// TIA Portal V17 export
// export: Created 2025-03-05T07:59:49.5409179Z, ExportSetting WithDefaults, DisplayName Totally Integrated Automation Portal, DisplayVersion V17 Update 8, DisplayName TIA Portal Openness, DisplayVersion V17 Update 8, DisplayName TIA Portal Version Control Interface, DisplayVersion V17, DisplayName SINAMICS Startdrive Advanced, DisplayVersion V17 SP2, DisplayName SINAMICS Startdrive G110M, G120, G120C, G120D, G120P, G115D, DisplayVersion V17 SP2, DisplayName SINAMICS Startdrive G130, G150, S120, S150, SINAMICS MV, S210, DisplayVersion V17 SP2, DisplayName STEP 7 Professional, DisplayVersion V17 Update 8, DisplayName SINUMERIK ONE STEP 7 Toolbox, DisplayVersion V17 Update 12, DisplayName SINUMERIK 840D sl STEP 7 Toolbox, DisplayVersion V17 Update 12, DisplayName STEP 7 Safety, DisplayVersion V17 Update 6, DisplayName WinCC Advanced, DisplayVersion V17 Update 8
FUNCTION "FC368_NCK_M_CH8_UNIT_03" : Void   // FC368, LAD
TITLE = Channel 1 data
{ S7_Optimized_Access := 'FALSE' }
AUTHOR : ETXETAR
VERSION : 1.0
// stored: AutoNumber false, IsIECCheckEnabled false, SetENOAutomatically false, UDAEnableTagReadback false
   VAR_TEMP
      auxm3 : Bool;
      auxm5 : Bool;
   END_VAR
   VAR_TEMP   // added for the SCL form of the ladder/FBD networks
      _w1 : Bool;
      _w2 : Bool;
   END_VAR
BEGIN

REGION Network 1: CALL FB331 M CODE EXTENDED CH4 / M CODE EXTENDED CHANNEL 2
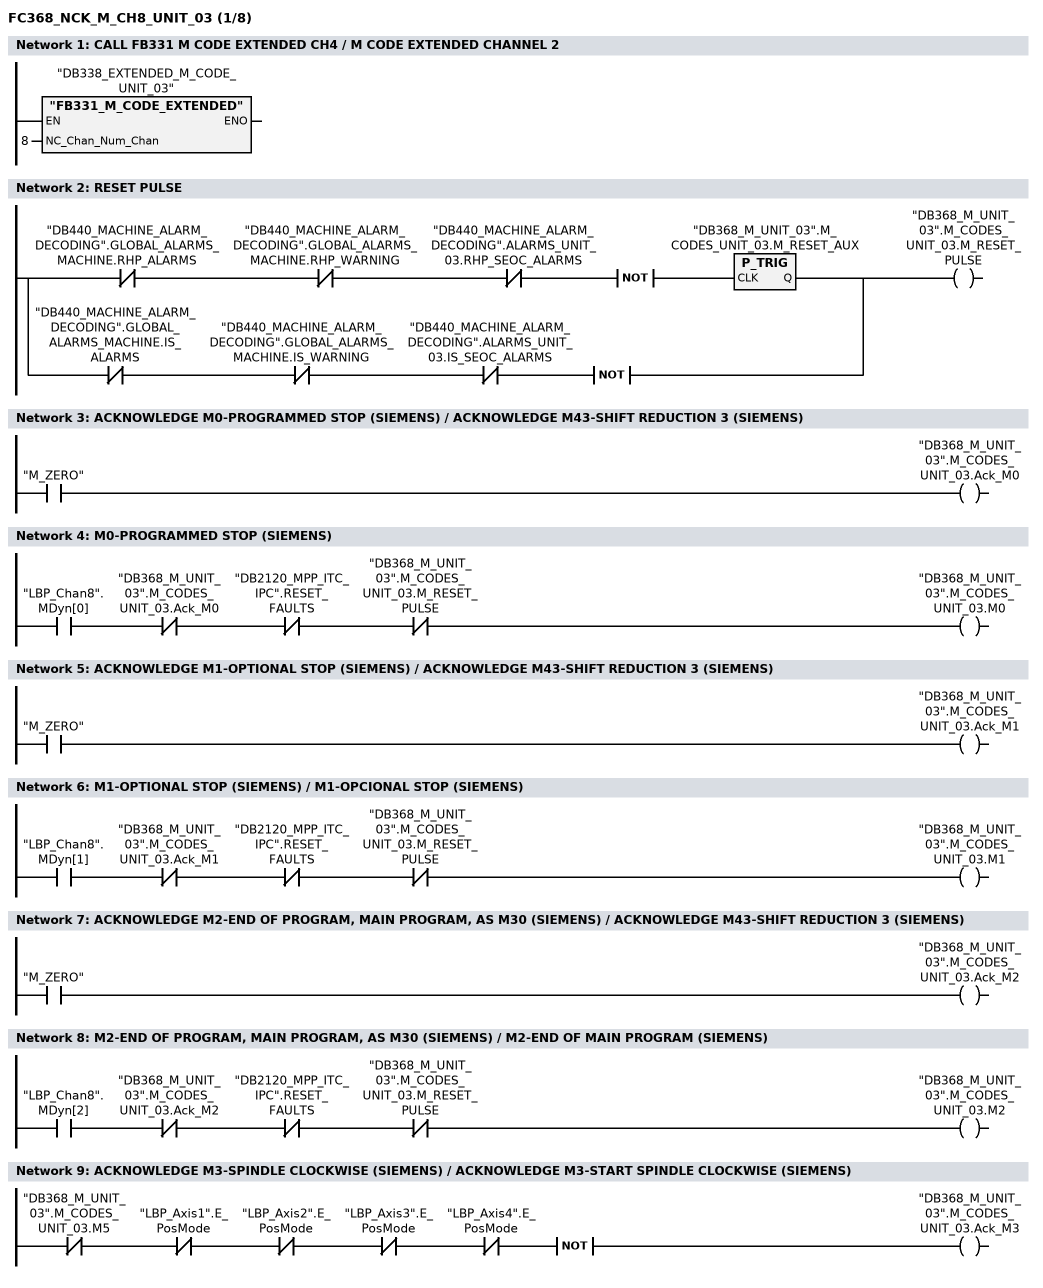
   RUNG wire#powerrail
      "DB338_EXTENDED_M_CODE_UNIT_03"(NC_Chan_Num_Chan := 8)
   END_RUNG
   // the same network as SCL:
   "DB338_EXTENDED_M_CODE_UNIT_03"(NC_Chan_Num_Chan := 8);   // "FB331_M_CODE_EXTENDED"
END_REGION

REGION Network 2: RESET PULSE
   RUNG wire#powerrail
      I_Contact( "DB440_MACHINE_ALARM_DECODING".GLOBAL_ALARMS_MACHINE.RHP_ALARMS )
      I_Contact( "DB440_MACHINE_ALARM_DECODING".GLOBAL_ALARMS_MACHINE.RHP_WARNING )
      I_Contact( "DB440_MACHINE_ALARM_DECODING".ALARMS_UNIT_03.RHP_SEOC_ALARMS )
      Not()
      P_Trig( "DB368_M_UNIT_03".M_CODES_UNIT_03.M_RESET_AUX )
      wire#w1
      Coil( "DB368_M_UNIT_03".M_CODES_UNIT_03.M_RESET_PULSE )
   END_RUNG
   RUNG wire#powerrail
      I_Contact( "DB440_MACHINE_ALARM_DECODING".GLOBAL_ALARMS_MACHINE.IS_ALARMS )
      I_Contact( "DB440_MACHINE_ALARM_DECODING".GLOBAL_ALARMS_MACHINE.IS_WARNING )
      I_Contact( "DB440_MACHINE_ALARM_DECODING".ALARMS_UNIT_03.IS_SEOC_ALARMS )
      Not()
   END_RUNG wire#w1
   // the same network as SCL:
   #_w1 := NOT (NOT "DB440_MACHINE_ALARM_DECODING".GLOBAL_ALARMS_MACHINE.RHP_ALARMS AND NOT "DB440_MACHINE_ALARM_DECODING".GLOBAL_ALARMS_MACHINE.RHP_WARNING AND NOT "DB440_MACHINE_ALARM_DECODING".ALARMS_UNIT_03.RHP_SEOC_ALARMS);
   #_w2 := #_w1 AND NOT "DB368_M_UNIT_03".M_CODES_UNIT_03.M_RESET_AUX;   // rising edge
   "DB368_M_UNIT_03".M_CODES_UNIT_03.M_RESET_AUX := #_w1;
   "DB368_M_UNIT_03".M_CODES_UNIT_03.M_RESET_PULSE := #_w2 OR NOT (NOT "DB440_MACHINE_ALARM_DECODING".GLOBAL_ALARMS_MACHINE.IS_ALARMS AND NOT "DB440_MACHINE_ALARM_DECODING".GLOBAL_ALARMS_MACHINE.IS_WARNING AND NOT "DB440_MACHINE_ALARM_DECODING".ALARMS_UNIT_03.IS_SEOC_ALARMS);
END_REGION

REGION Network 3: ACKNOWLEDGE M0-PROGRAMMED STOP (SIEMENS) / ACKNOWLEDGE M43-SHIFT REDUCTION 3 (SIEMENS)
   RUNG wire#powerrail
      Contact( "M_ZERO" )
      Coil( "DB368_M_UNIT_03".M_CODES_UNIT_03.Ack_M0 )
   END_RUNG
   // the same network as SCL:
   "DB368_M_UNIT_03".M_CODES_UNIT_03.Ack_M0 := "M_ZERO";
END_REGION

REGION Network 4: M0-PROGRAMMED STOP (SIEMENS)
   RUNG wire#powerrail
      Contact( "LBP_Chan8".MDyn[0] )
      I_Contact( "DB368_M_UNIT_03".M_CODES_UNIT_03.Ack_M0 )
      I_Contact( "DB2120_MPP_ITC_IPC".RESET_FAULTS )
      I_Contact( "DB368_M_UNIT_03".M_CODES_UNIT_03.M_RESET_PULSE )
      Coil( "DB368_M_UNIT_03".M_CODES_UNIT_03.M0 )
   END_RUNG
   // the same network as SCL:
   "DB368_M_UNIT_03".M_CODES_UNIT_03.M0 := "LBP_Chan8".MDyn[0] AND NOT "DB368_M_UNIT_03".M_CODES_UNIT_03.Ack_M0 AND NOT "DB2120_MPP_ITC_IPC".RESET_FAULTS AND NOT "DB368_M_UNIT_03".M_CODES_UNIT_03.M_RESET_PULSE;
END_REGION

REGION Network 5: ACKNOWLEDGE M1-OPTIONAL STOP (SIEMENS) / ACKNOWLEDGE M43-SHIFT REDUCTION 3 (SIEMENS)
   RUNG wire#powerrail
      Contact( "M_ZERO" )
      Coil( "DB368_M_UNIT_03".M_CODES_UNIT_03.Ack_M1 )
   END_RUNG
   // the same network as SCL:
   "DB368_M_UNIT_03".M_CODES_UNIT_03.Ack_M1 := "M_ZERO";
END_REGION

REGION Network 6: M1-OPTIONAL STOP (SIEMENS) / M1-OPCIONAL STOP (SIEMENS)
   RUNG wire#powerrail
      Contact( "LBP_Chan8".MDyn[1] )
      I_Contact( "DB368_M_UNIT_03".M_CODES_UNIT_03.Ack_M1 )
      I_Contact( "DB2120_MPP_ITC_IPC".RESET_FAULTS )
      I_Contact( "DB368_M_UNIT_03".M_CODES_UNIT_03.M_RESET_PULSE )
      Coil( "DB368_M_UNIT_03".M_CODES_UNIT_03.M1 )
   END_RUNG
   // the same network as SCL:
   "DB368_M_UNIT_03".M_CODES_UNIT_03.M1 := "LBP_Chan8".MDyn[1] AND NOT "DB368_M_UNIT_03".M_CODES_UNIT_03.Ack_M1 AND NOT "DB2120_MPP_ITC_IPC".RESET_FAULTS AND NOT "DB368_M_UNIT_03".M_CODES_UNIT_03.M_RESET_PULSE;
END_REGION

REGION Network 7: ACKNOWLEDGE M2-END OF PROGRAM, MAIN PROGRAM, AS M30 (SIEMENS) / ACKNOWLEDGE M43-SHIFT REDUCTION 3 (SIEMENS)
   RUNG wire#powerrail
      Contact( "M_ZERO" )
      Coil( "DB368_M_UNIT_03".M_CODES_UNIT_03.Ack_M2 )
   END_RUNG
   // the same network as SCL:
   "DB368_M_UNIT_03".M_CODES_UNIT_03.Ack_M2 := "M_ZERO";
END_REGION

REGION Network 8: M2-END OF PROGRAM, MAIN PROGRAM, AS M30 (SIEMENS) / M2-END OF MAIN PROGRAM (SIEMENS)
   RUNG wire#powerrail
      Contact( "LBP_Chan8".MDyn[2] )
      I_Contact( "DB368_M_UNIT_03".M_CODES_UNIT_03.Ack_M2 )
      I_Contact( "DB2120_MPP_ITC_IPC".RESET_FAULTS )
      I_Contact( "DB368_M_UNIT_03".M_CODES_UNIT_03.M_RESET_PULSE )
      Coil( "DB368_M_UNIT_03".M_CODES_UNIT_03.M2 )
   END_RUNG
   // the same network as SCL:
   "DB368_M_UNIT_03".M_CODES_UNIT_03.M2 := "LBP_Chan8".MDyn[2] AND NOT "DB368_M_UNIT_03".M_CODES_UNIT_03.Ack_M2 AND NOT "DB2120_MPP_ITC_IPC".RESET_FAULTS AND NOT "DB368_M_UNIT_03".M_CODES_UNIT_03.M_RESET_PULSE;
END_REGION

REGION Network 9: ACKNOWLEDGE M3-SPINDLE CLOCKWISE (SIEMENS) / ACKNOWLEDGE M3-START SPINDLE CLOCKWISE (SIEMENS)
   RUNG wire#powerrail
      I_Contact( "DB368_M_UNIT_03".M_CODES_UNIT_03.M5 )
      I_Contact( "LBP_Axis1".E_PosMode )
      I_Contact( "LBP_Axis2".E_PosMode )
      I_Contact( "LBP_Axis3".E_PosMode )
      I_Contact( "LBP_Axis4".E_PosMode )
      Not()
      Coil( "DB368_M_UNIT_03".M_CODES_UNIT_03.Ack_M3 )
   END_RUNG
   // the same network as SCL:
   "DB368_M_UNIT_03".M_CODES_UNIT_03.Ack_M3 := NOT (NOT "DB368_M_UNIT_03".M_CODES_UNIT_03.M5 AND NOT "LBP_Axis1".E_PosMode AND NOT "LBP_Axis2".E_PosMode AND NOT "LBP_Axis3".E_PosMode AND NOT "LBP_Axis4".E_PosMode);
END_REGION

REGION Network 10: M3-SPINDLE CLOCKWISE AUXILIARY (SIEMENS) / Extended address M function 1 (16 bit INT)
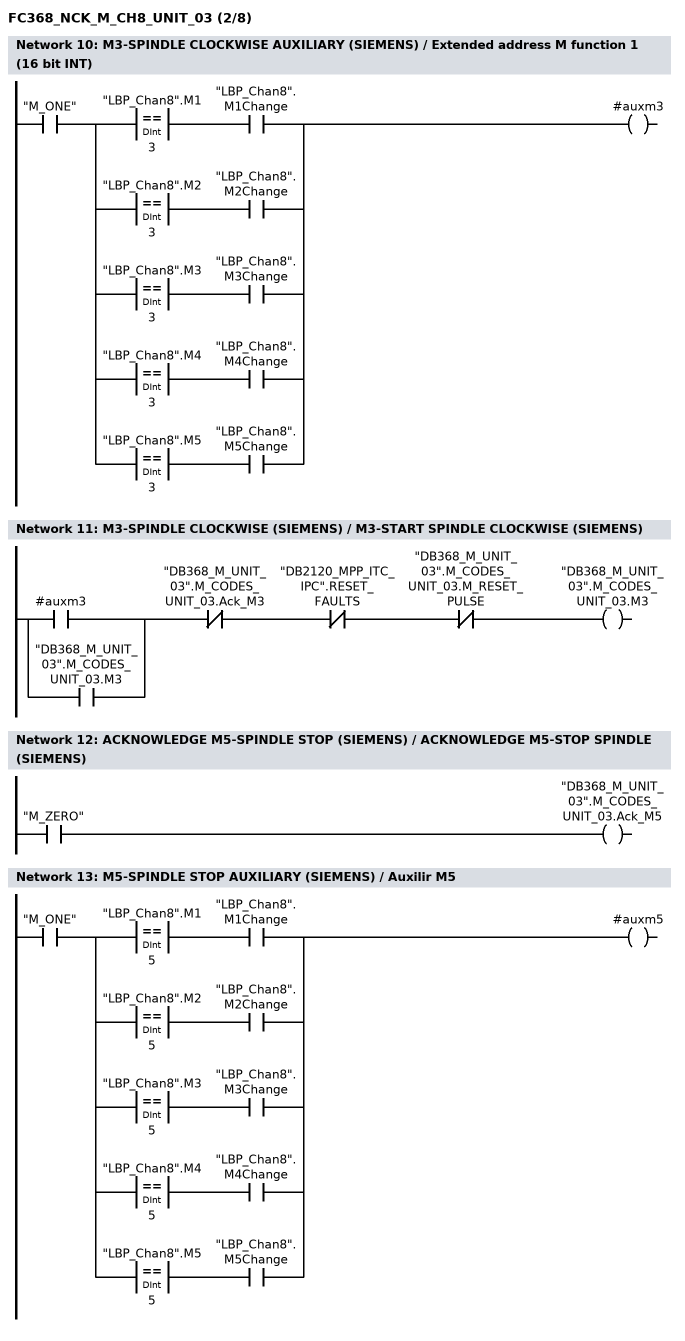
   RUNG wire#powerrail
      Contact( "M_ONE" )
      wire#w1
      { S7_Templates := "SrcType := DInt" } EQ_Contact(in1 := "LBP_Chan8".M1, in2 := 3)
      Contact( "LBP_Chan8".M1Change )
      wire#w2
      Coil( #auxm3 )
   END_RUNG
   RUNG wire#w1
      { S7_Templates := "SrcType := DInt" } EQ_Contact(in1 := "LBP_Chan8".M2, in2 := 3)
      Contact( "LBP_Chan8".M2Change )
   END_RUNG wire#w2
   RUNG wire#w1
      { S7_Templates := "SrcType := DInt" } EQ_Contact(in1 := "LBP_Chan8".M3, in2 := 3)
      Contact( "LBP_Chan8".M3Change )
   END_RUNG wire#w2
   RUNG wire#w1
      { S7_Templates := "SrcType := DInt" } EQ_Contact(in1 := "LBP_Chan8".M4, in2 := 3)
      Contact( "LBP_Chan8".M4Change )
   END_RUNG wire#w2
   RUNG wire#w1
      { S7_Templates := "SrcType := DInt" } EQ_Contact(in1 := "LBP_Chan8".M5, in2 := 3)
      Contact( "LBP_Chan8".M5Change )
   END_RUNG wire#w2
   // the same network as SCL:
   #auxm3 := "M_ONE" AND ((("LBP_Chan8".M1 = 3) AND "LBP_Chan8".M1Change) OR (("LBP_Chan8".M2 = 3) AND "LBP_Chan8".M2Change) OR (("LBP_Chan8".M3 = 3) AND "LBP_Chan8".M3Change) OR (("LBP_Chan8".M4 = 3) AND "LBP_Chan8".M4Change) OR (("LBP_Chan8".M5 = 3) AND "LBP_Chan8".M5Change));
END_REGION

REGION Network 11: M3-SPINDLE CLOCKWISE (SIEMENS) / M3-START SPINDLE CLOCKWISE (SIEMENS)
   RUNG wire#powerrail
      Contact( #auxm3 )
      wire#w1
      I_Contact( "DB368_M_UNIT_03".M_CODES_UNIT_03.Ack_M3 )
      I_Contact( "DB2120_MPP_ITC_IPC".RESET_FAULTS )
      I_Contact( "DB368_M_UNIT_03".M_CODES_UNIT_03.M_RESET_PULSE )
      Coil( "DB368_M_UNIT_03".M_CODES_UNIT_03.M3 )
   END_RUNG
   RUNG wire#powerrail
      Contact( "DB368_M_UNIT_03".M_CODES_UNIT_03.M3 )
   END_RUNG wire#w1
   // the same network as SCL:
   "DB368_M_UNIT_03".M_CODES_UNIT_03.M3 := (#auxm3 OR "DB368_M_UNIT_03".M_CODES_UNIT_03.M3) AND NOT "DB368_M_UNIT_03".M_CODES_UNIT_03.Ack_M3 AND NOT "DB2120_MPP_ITC_IPC".RESET_FAULTS AND NOT "DB368_M_UNIT_03".M_CODES_UNIT_03.M_RESET_PULSE;
END_REGION

REGION Network 12: ACKNOWLEDGE M5-SPINDLE STOP (SIEMENS) / ACKNOWLEDGE M5-STOP SPINDLE (SIEMENS)
   RUNG wire#powerrail
      Contact( "M_ZERO" )
      Coil( "DB368_M_UNIT_03".M_CODES_UNIT_03.Ack_M5 )
   END_RUNG
   // the same network as SCL:
   "DB368_M_UNIT_03".M_CODES_UNIT_03.Ack_M5 := "M_ZERO";
END_REGION

REGION Network 13: M5-SPINDLE STOP AUXILIARY (SIEMENS) / Auxilir M5
   RUNG wire#powerrail
      Contact( "M_ONE" )
      wire#w1
      { S7_Templates := "SrcType := DInt" } EQ_Contact(in1 := "LBP_Chan8".M1, in2 := 5)
      Contact( "LBP_Chan8".M1Change )
      wire#w2
      Coil( #auxm5 )
   END_RUNG
   RUNG wire#w1
      { S7_Templates := "SrcType := DInt" } EQ_Contact(in1 := "LBP_Chan8".M2, in2 := 5)
      Contact( "LBP_Chan8".M2Change )
   END_RUNG wire#w2
   RUNG wire#w1
      { S7_Templates := "SrcType := DInt" } EQ_Contact(in1 := "LBP_Chan8".M3, in2 := 5)
      Contact( "LBP_Chan8".M3Change )
   END_RUNG wire#w2
   RUNG wire#w1
      { S7_Templates := "SrcType := DInt" } EQ_Contact(in1 := "LBP_Chan8".M4, in2 := 5)
      Contact( "LBP_Chan8".M4Change )
   END_RUNG wire#w2
   RUNG wire#w1
      { S7_Templates := "SrcType := DInt" } EQ_Contact(in1 := "LBP_Chan8".M5, in2 := 5)
      Contact( "LBP_Chan8".M5Change )
   END_RUNG wire#w2
   // the same network as SCL:
   #auxm5 := "M_ONE" AND ((("LBP_Chan8".M1 = 5) AND "LBP_Chan8".M1Change) OR (("LBP_Chan8".M2 = 5) AND "LBP_Chan8".M2Change) OR (("LBP_Chan8".M3 = 5) AND "LBP_Chan8".M3Change) OR (("LBP_Chan8".M4 = 5) AND "LBP_Chan8".M4Change) OR (("LBP_Chan8".M5 = 5) AND "LBP_Chan8".M5Change));
END_REGION

REGION Network 14: M5-SPINDLE STOP (SIEMENS) / M5-STOP SPINDLE (SIEMENS)
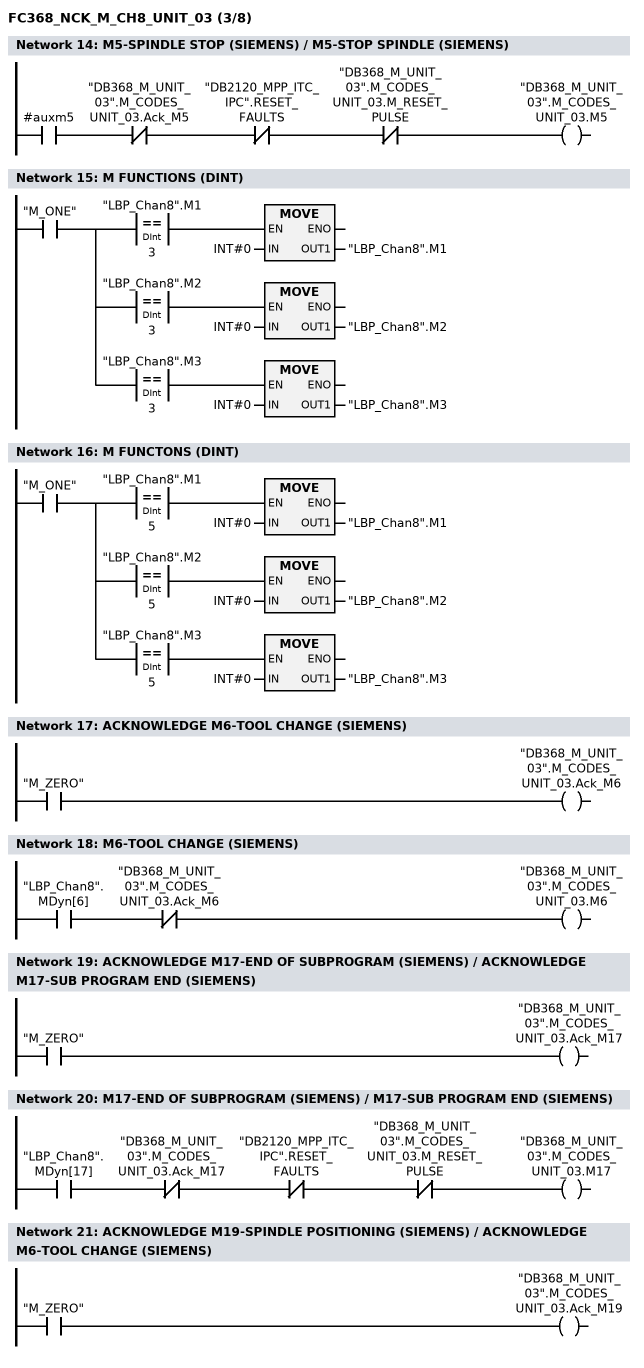
   RUNG wire#powerrail
      Contact( #auxm5 )
      I_Contact( "DB368_M_UNIT_03".M_CODES_UNIT_03.Ack_M5 )
      I_Contact( "DB2120_MPP_ITC_IPC".RESET_FAULTS )
      I_Contact( "DB368_M_UNIT_03".M_CODES_UNIT_03.M_RESET_PULSE )
      Coil( "DB368_M_UNIT_03".M_CODES_UNIT_03.M5 )
   END_RUNG
   // the same network as SCL:
   "DB368_M_UNIT_03".M_CODES_UNIT_03.M5 := #auxm5 AND NOT "DB368_M_UNIT_03".M_CODES_UNIT_03.Ack_M5 AND NOT "DB2120_MPP_ITC_IPC".RESET_FAULTS AND NOT "DB368_M_UNIT_03".M_CODES_UNIT_03.M_RESET_PULSE;
END_REGION

REGION Network 15: M FUNCTIONS (DINT)
   RUNG wire#powerrail
      Contact( "M_ONE" )
      wire#w1
      { S7_Templates := "SrcType := DInt" } EQ_Contact(in1 := "LBP_Chan8".M1, in2 := 3)
      { S7_GenerateENO := "TRUE" } Move(in := INT#0, out1 => "LBP_Chan8".M1)
   END_RUNG
   RUNG wire#w1
      { S7_Templates := "SrcType := DInt" } EQ_Contact(in1 := "LBP_Chan8".M2, in2 := 3)
      { S7_GenerateENO := "TRUE" } Move(in := INT#0, out1 => "LBP_Chan8".M2)
   END_RUNG
   RUNG wire#w1
      { S7_Templates := "SrcType := DInt" } EQ_Contact(in1 := "LBP_Chan8".M3, in2 := 3)
      { S7_GenerateENO := "TRUE" } Move(in := INT#0, out1 => "LBP_Chan8".M3)
   END_RUNG
   // the same network as SCL:
   IF "M_ONE" AND ("LBP_Chan8".M1 = 3) THEN "LBP_Chan8".M1 := INT#0; END_IF;
   IF "M_ONE" AND ("LBP_Chan8".M2 = 3) THEN "LBP_Chan8".M2 := INT#0; END_IF;
   IF "M_ONE" AND ("LBP_Chan8".M3 = 3) THEN "LBP_Chan8".M3 := INT#0; END_IF;
END_REGION

REGION Network 16: M FUNCTONS (DINT)
   RUNG wire#powerrail
      Contact( "M_ONE" )
      wire#w1
      { S7_Templates := "SrcType := DInt" } EQ_Contact(in1 := "LBP_Chan8".M1, in2 := 5)
      { S7_GenerateENO := "TRUE" } Move(in := INT#0, out1 => "LBP_Chan8".M1)
   END_RUNG
   RUNG wire#w1
      { S7_Templates := "SrcType := DInt" } EQ_Contact(in1 := "LBP_Chan8".M2, in2 := 5)
      { S7_GenerateENO := "TRUE" } Move(in := INT#0, out1 => "LBP_Chan8".M2)
   END_RUNG
   RUNG wire#w1
      { S7_Templates := "SrcType := DInt" } EQ_Contact(in1 := "LBP_Chan8".M3, in2 := 5)
      { S7_GenerateENO := "TRUE" } Move(in := INT#0, out1 => "LBP_Chan8".M3)
   END_RUNG
   // the same network as SCL:
   IF "M_ONE" AND ("LBP_Chan8".M1 = 5) THEN "LBP_Chan8".M1 := INT#0; END_IF;
   IF "M_ONE" AND ("LBP_Chan8".M2 = 5) THEN "LBP_Chan8".M2 := INT#0; END_IF;
   IF "M_ONE" AND ("LBP_Chan8".M3 = 5) THEN "LBP_Chan8".M3 := INT#0; END_IF;
END_REGION

REGION Network 17: ACKNOWLEDGE M6-TOOL CHANGE (SIEMENS)
   RUNG wire#powerrail
      Contact( "M_ZERO" )
      Coil( "DB368_M_UNIT_03".M_CODES_UNIT_03.Ack_M6 )
   END_RUNG
   // the same network as SCL:
   "DB368_M_UNIT_03".M_CODES_UNIT_03.Ack_M6 := "M_ZERO";
END_REGION

REGION Network 18: M6-TOOL CHANGE (SIEMENS)
   RUNG wire#powerrail
      Contact( "LBP_Chan8".MDyn[6] )
      I_Contact( "DB368_M_UNIT_03".M_CODES_UNIT_03.Ack_M6 )
      Coil( "DB368_M_UNIT_03".M_CODES_UNIT_03.M6 )
   END_RUNG
   // the same network as SCL:
   "DB368_M_UNIT_03".M_CODES_UNIT_03.M6 := "LBP_Chan8".MDyn[6] AND NOT "DB368_M_UNIT_03".M_CODES_UNIT_03.Ack_M6;
END_REGION

REGION Network 19: ACKNOWLEDGE M17-END OF SUBPROGRAM (SIEMENS) / ACKNOWLEDGE M17-SUB PROGRAM END (SIEMENS)
   RUNG wire#powerrail
      Contact( "M_ZERO" )
      Coil( "DB368_M_UNIT_03".M_CODES_UNIT_03.Ack_M17 )
   END_RUNG
   // the same network as SCL:
   "DB368_M_UNIT_03".M_CODES_UNIT_03.Ack_M17 := "M_ZERO";
END_REGION

REGION Network 20: M17-END OF SUBPROGRAM (SIEMENS) / M17-SUB PROGRAM END (SIEMENS)
   RUNG wire#powerrail
      Contact( "LBP_Chan8".MDyn[17] )
      I_Contact( "DB368_M_UNIT_03".M_CODES_UNIT_03.Ack_M17 )
      I_Contact( "DB2120_MPP_ITC_IPC".RESET_FAULTS )
      I_Contact( "DB368_M_UNIT_03".M_CODES_UNIT_03.M_RESET_PULSE )
      Coil( "DB368_M_UNIT_03".M_CODES_UNIT_03.M17 )
   END_RUNG
   // the same network as SCL:
   "DB368_M_UNIT_03".M_CODES_UNIT_03.M17 := "LBP_Chan8".MDyn[17] AND NOT "DB368_M_UNIT_03".M_CODES_UNIT_03.Ack_M17 AND NOT "DB2120_MPP_ITC_IPC".RESET_FAULTS AND NOT "DB368_M_UNIT_03".M_CODES_UNIT_03.M_RESET_PULSE;
END_REGION

REGION Network 21: ACKNOWLEDGE M19-SPINDLE POSITIONING (SIEMENS) / ACKNOWLEDGE M6-TOOL CHANGE (SIEMENS)
   RUNG wire#powerrail
      Contact( "M_ZERO" )
      Coil( "DB368_M_UNIT_03".M_CODES_UNIT_03.Ack_M19 )
   END_RUNG
   // the same network as SCL:
   "DB368_M_UNIT_03".M_CODES_UNIT_03.Ack_M19 := "M_ZERO";
END_REGION

REGION Network 22: M19-SPINDLE POSITIONING (SIEMENS) / M6-TOOL CHANGE (SIEMENS)
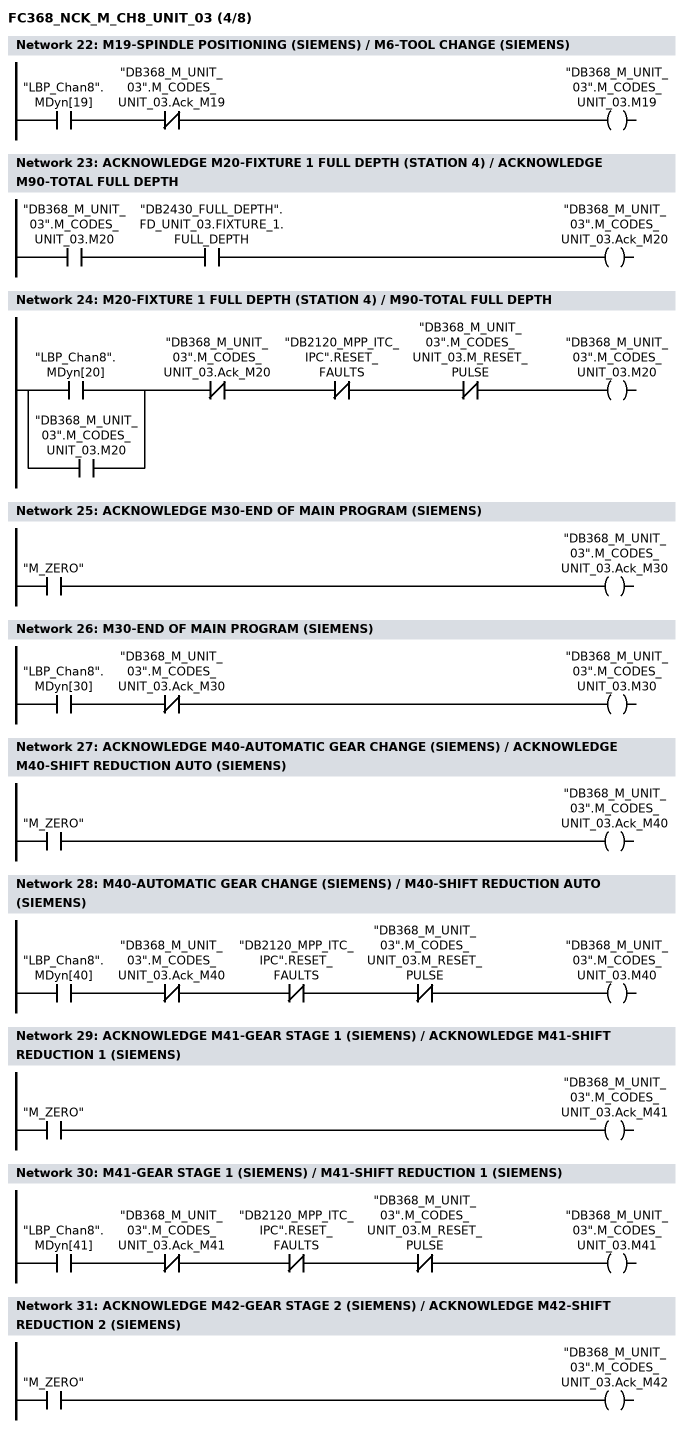
   RUNG wire#powerrail
      Contact( "LBP_Chan8".MDyn[19] )
      I_Contact( "DB368_M_UNIT_03".M_CODES_UNIT_03.Ack_M19 )
      Coil( "DB368_M_UNIT_03".M_CODES_UNIT_03.M19 )
   END_RUNG
   // the same network as SCL:
   "DB368_M_UNIT_03".M_CODES_UNIT_03.M19 := "LBP_Chan8".MDyn[19] AND NOT "DB368_M_UNIT_03".M_CODES_UNIT_03.Ack_M19;
END_REGION

REGION Network 23: ACKNOWLEDGE M20-FIXTURE 1 FULL DEPTH (STATION 4) / ACKNOWLEDGE M90-TOTAL FULL DEPTH
   RUNG wire#powerrail
      Contact( "DB368_M_UNIT_03".M_CODES_UNIT_03.M20 )
      Contact( "DB2430_FULL_DEPTH".FD_UNIT_03.FIXTURE_1.FULL_DEPTH )
      Coil( "DB368_M_UNIT_03".M_CODES_UNIT_03.Ack_M20 )
   END_RUNG
   // the same network as SCL:
   "DB368_M_UNIT_03".M_CODES_UNIT_03.Ack_M20 := "DB368_M_UNIT_03".M_CODES_UNIT_03.M20 AND "DB2430_FULL_DEPTH".FD_UNIT_03.FIXTURE_1.FULL_DEPTH;
END_REGION

REGION Network 24: M20-FIXTURE 1 FULL DEPTH (STATION 4) / M90-TOTAL FULL DEPTH
   RUNG wire#powerrail
      Contact( "LBP_Chan8".MDyn[20] )
      wire#w1
      I_Contact( "DB368_M_UNIT_03".M_CODES_UNIT_03.Ack_M20 )
      I_Contact( "DB2120_MPP_ITC_IPC".RESET_FAULTS )
      I_Contact( "DB368_M_UNIT_03".M_CODES_UNIT_03.M_RESET_PULSE )
      Coil( "DB368_M_UNIT_03".M_CODES_UNIT_03.M20 )
   END_RUNG
   RUNG wire#powerrail
      Contact( "DB368_M_UNIT_03".M_CODES_UNIT_03.M20 )
   END_RUNG wire#w1
   // the same network as SCL:
   "DB368_M_UNIT_03".M_CODES_UNIT_03.M20 := ("LBP_Chan8".MDyn[20] OR "DB368_M_UNIT_03".M_CODES_UNIT_03.M20) AND NOT "DB368_M_UNIT_03".M_CODES_UNIT_03.Ack_M20 AND NOT "DB2120_MPP_ITC_IPC".RESET_FAULTS AND NOT "DB368_M_UNIT_03".M_CODES_UNIT_03.M_RESET_PULSE;
END_REGION

REGION Network 25: ACKNOWLEDGE M30-END OF MAIN PROGRAM (SIEMENS)
   RUNG wire#powerrail
      Contact( "M_ZERO" )
      Coil( "DB368_M_UNIT_03".M_CODES_UNIT_03.Ack_M30 )
   END_RUNG
   // the same network as SCL:
   "DB368_M_UNIT_03".M_CODES_UNIT_03.Ack_M30 := "M_ZERO";
END_REGION

REGION Network 26: M30-END OF MAIN PROGRAM (SIEMENS)
   RUNG wire#powerrail
      Contact( "LBP_Chan8".MDyn[30] )
      I_Contact( "DB368_M_UNIT_03".M_CODES_UNIT_03.Ack_M30 )
      Coil( "DB368_M_UNIT_03".M_CODES_UNIT_03.M30 )
   END_RUNG
   // the same network as SCL:
   "DB368_M_UNIT_03".M_CODES_UNIT_03.M30 := "LBP_Chan8".MDyn[30] AND NOT "DB368_M_UNIT_03".M_CODES_UNIT_03.Ack_M30;
END_REGION

REGION Network 27: ACKNOWLEDGE M40-AUTOMATIC GEAR CHANGE (SIEMENS) / ACKNOWLEDGE M40-SHIFT REDUCTION AUTO (SIEMENS)
   RUNG wire#powerrail
      Contact( "M_ZERO" )
      Coil( "DB368_M_UNIT_03".M_CODES_UNIT_03.Ack_M40 )
   END_RUNG
   // the same network as SCL:
   "DB368_M_UNIT_03".M_CODES_UNIT_03.Ack_M40 := "M_ZERO";
END_REGION

REGION Network 28: M40-AUTOMATIC GEAR CHANGE (SIEMENS) / M40-SHIFT REDUCTION AUTO (SIEMENS)
   RUNG wire#powerrail
      Contact( "LBP_Chan8".MDyn[40] )
      I_Contact( "DB368_M_UNIT_03".M_CODES_UNIT_03.Ack_M40 )
      I_Contact( "DB2120_MPP_ITC_IPC".RESET_FAULTS )
      I_Contact( "DB368_M_UNIT_03".M_CODES_UNIT_03.M_RESET_PULSE )
      Coil( "DB368_M_UNIT_03".M_CODES_UNIT_03.M40 )
   END_RUNG
   // the same network as SCL:
   "DB368_M_UNIT_03".M_CODES_UNIT_03.M40 := "LBP_Chan8".MDyn[40] AND NOT "DB368_M_UNIT_03".M_CODES_UNIT_03.Ack_M40 AND NOT "DB2120_MPP_ITC_IPC".RESET_FAULTS AND NOT "DB368_M_UNIT_03".M_CODES_UNIT_03.M_RESET_PULSE;
END_REGION

REGION Network 29: ACKNOWLEDGE M41-GEAR STAGE 1 (SIEMENS) / ACKNOWLEDGE M41-SHIFT REDUCTION 1 (SIEMENS)
   RUNG wire#powerrail
      Contact( "M_ZERO" )
      Coil( "DB368_M_UNIT_03".M_CODES_UNIT_03.Ack_M41 )
   END_RUNG
   // the same network as SCL:
   "DB368_M_UNIT_03".M_CODES_UNIT_03.Ack_M41 := "M_ZERO";
END_REGION

REGION Network 30: M41-GEAR STAGE 1 (SIEMENS) / M41-SHIFT REDUCTION 1 (SIEMENS)
   RUNG wire#powerrail
      Contact( "LBP_Chan8".MDyn[41] )
      I_Contact( "DB368_M_UNIT_03".M_CODES_UNIT_03.Ack_M41 )
      I_Contact( "DB2120_MPP_ITC_IPC".RESET_FAULTS )
      I_Contact( "DB368_M_UNIT_03".M_CODES_UNIT_03.M_RESET_PULSE )
      Coil( "DB368_M_UNIT_03".M_CODES_UNIT_03.M41 )
   END_RUNG
   // the same network as SCL:
   "DB368_M_UNIT_03".M_CODES_UNIT_03.M41 := "LBP_Chan8".MDyn[41] AND NOT "DB368_M_UNIT_03".M_CODES_UNIT_03.Ack_M41 AND NOT "DB2120_MPP_ITC_IPC".RESET_FAULTS AND NOT "DB368_M_UNIT_03".M_CODES_UNIT_03.M_RESET_PULSE;
END_REGION

REGION Network 31: ACKNOWLEDGE M42-GEAR STAGE 2 (SIEMENS) / ACKNOWLEDGE M42-SHIFT REDUCTION 2 (SIEMENS)
   RUNG wire#powerrail
      Contact( "M_ZERO" )
      Coil( "DB368_M_UNIT_03".M_CODES_UNIT_03.Ack_M42 )
   END_RUNG
   // the same network as SCL:
   "DB368_M_UNIT_03".M_CODES_UNIT_03.Ack_M42 := "M_ZERO";
END_REGION

REGION Network 32: M42-GEAR STAGE 2 (SIEMENS) / M42-SHIFT REDUCTION 2 (SIEMENS)
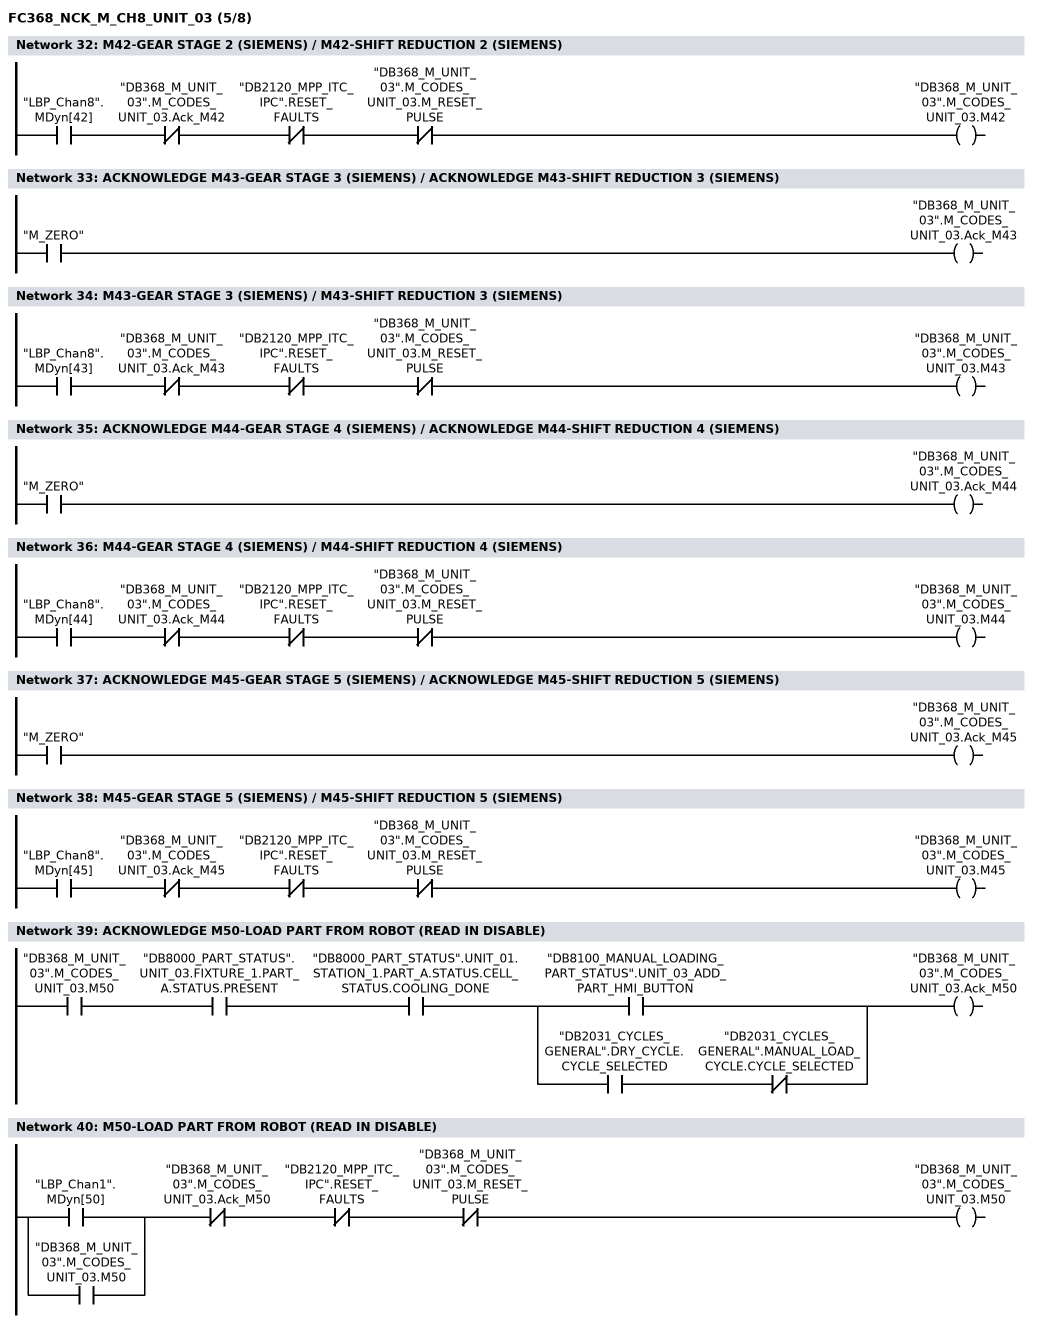
   RUNG wire#powerrail
      Contact( "LBP_Chan8".MDyn[42] )
      I_Contact( "DB368_M_UNIT_03".M_CODES_UNIT_03.Ack_M42 )
      I_Contact( "DB2120_MPP_ITC_IPC".RESET_FAULTS )
      I_Contact( "DB368_M_UNIT_03".M_CODES_UNIT_03.M_RESET_PULSE )
      Coil( "DB368_M_UNIT_03".M_CODES_UNIT_03.M42 )
   END_RUNG
   // the same network as SCL:
   "DB368_M_UNIT_03".M_CODES_UNIT_03.M42 := "LBP_Chan8".MDyn[42] AND NOT "DB368_M_UNIT_03".M_CODES_UNIT_03.Ack_M42 AND NOT "DB2120_MPP_ITC_IPC".RESET_FAULTS AND NOT "DB368_M_UNIT_03".M_CODES_UNIT_03.M_RESET_PULSE;
END_REGION

REGION Network 33: ACKNOWLEDGE M43-GEAR STAGE 3 (SIEMENS) / ACKNOWLEDGE M43-SHIFT REDUCTION 3 (SIEMENS)
   RUNG wire#powerrail
      Contact( "M_ZERO" )
      Coil( "DB368_M_UNIT_03".M_CODES_UNIT_03.Ack_M43 )
   END_RUNG
   // the same network as SCL:
   "DB368_M_UNIT_03".M_CODES_UNIT_03.Ack_M43 := "M_ZERO";
END_REGION

REGION Network 34: M43-GEAR STAGE 3 (SIEMENS) / M43-SHIFT REDUCTION 3 (SIEMENS)
   RUNG wire#powerrail
      Contact( "LBP_Chan8".MDyn[43] )
      I_Contact( "DB368_M_UNIT_03".M_CODES_UNIT_03.Ack_M43 )
      I_Contact( "DB2120_MPP_ITC_IPC".RESET_FAULTS )
      I_Contact( "DB368_M_UNIT_03".M_CODES_UNIT_03.M_RESET_PULSE )
      Coil( "DB368_M_UNIT_03".M_CODES_UNIT_03.M43 )
   END_RUNG
   // the same network as SCL:
   "DB368_M_UNIT_03".M_CODES_UNIT_03.M43 := "LBP_Chan8".MDyn[43] AND NOT "DB368_M_UNIT_03".M_CODES_UNIT_03.Ack_M43 AND NOT "DB2120_MPP_ITC_IPC".RESET_FAULTS AND NOT "DB368_M_UNIT_03".M_CODES_UNIT_03.M_RESET_PULSE;
END_REGION

REGION Network 35: ACKNOWLEDGE M44-GEAR STAGE 4 (SIEMENS) / ACKNOWLEDGE M44-SHIFT REDUCTION 4 (SIEMENS)
   RUNG wire#powerrail
      Contact( "M_ZERO" )
      Coil( "DB368_M_UNIT_03".M_CODES_UNIT_03.Ack_M44 )
   END_RUNG
   // the same network as SCL:
   "DB368_M_UNIT_03".M_CODES_UNIT_03.Ack_M44 := "M_ZERO";
END_REGION

REGION Network 36: M44-GEAR STAGE 4 (SIEMENS) / M44-SHIFT REDUCTION 4 (SIEMENS)
   RUNG wire#powerrail
      Contact( "LBP_Chan8".MDyn[44] )
      I_Contact( "DB368_M_UNIT_03".M_CODES_UNIT_03.Ack_M44 )
      I_Contact( "DB2120_MPP_ITC_IPC".RESET_FAULTS )
      I_Contact( "DB368_M_UNIT_03".M_CODES_UNIT_03.M_RESET_PULSE )
      Coil( "DB368_M_UNIT_03".M_CODES_UNIT_03.M44 )
   END_RUNG
   // the same network as SCL:
   "DB368_M_UNIT_03".M_CODES_UNIT_03.M44 := "LBP_Chan8".MDyn[44] AND NOT "DB368_M_UNIT_03".M_CODES_UNIT_03.Ack_M44 AND NOT "DB2120_MPP_ITC_IPC".RESET_FAULTS AND NOT "DB368_M_UNIT_03".M_CODES_UNIT_03.M_RESET_PULSE;
END_REGION

REGION Network 37: ACKNOWLEDGE M45-GEAR STAGE 5 (SIEMENS) / ACKNOWLEDGE M45-SHIFT REDUCTION 5 (SIEMENS)
   RUNG wire#powerrail
      Contact( "M_ZERO" )
      Coil( "DB368_M_UNIT_03".M_CODES_UNIT_03.Ack_M45 )
   END_RUNG
   // the same network as SCL:
   "DB368_M_UNIT_03".M_CODES_UNIT_03.Ack_M45 := "M_ZERO";
END_REGION

REGION Network 38: M45-GEAR STAGE 5 (SIEMENS) / M45-SHIFT REDUCTION 5 (SIEMENS)
   RUNG wire#powerrail
      Contact( "LBP_Chan8".MDyn[45] )
      I_Contact( "DB368_M_UNIT_03".M_CODES_UNIT_03.Ack_M45 )
      I_Contact( "DB2120_MPP_ITC_IPC".RESET_FAULTS )
      I_Contact( "DB368_M_UNIT_03".M_CODES_UNIT_03.M_RESET_PULSE )
      Coil( "DB368_M_UNIT_03".M_CODES_UNIT_03.M45 )
   END_RUNG
   // the same network as SCL:
   "DB368_M_UNIT_03".M_CODES_UNIT_03.M45 := "LBP_Chan8".MDyn[45] AND NOT "DB368_M_UNIT_03".M_CODES_UNIT_03.Ack_M45 AND NOT "DB2120_MPP_ITC_IPC".RESET_FAULTS AND NOT "DB368_M_UNIT_03".M_CODES_UNIT_03.M_RESET_PULSE;
END_REGION

REGION Network 39: ACKNOWLEDGE M50-LOAD PART FROM ROBOT (READ IN DISABLE)
   RUNG wire#powerrail
      Contact( "DB368_M_UNIT_03".M_CODES_UNIT_03.M50 )
      Contact( "DB8000_PART_STATUS".UNIT_03.FIXTURE_1.PART_A.STATUS.PRESENT )
      Contact( "DB8000_PART_STATUS".UNIT_01.STATION_1.PART_A.STATUS.CELL_STATUS.COOLING_DONE )
      wire#w1
      Contact( "DB8100_MANUAL_LOADING_PART_STATUS".UNIT_03_ADD_PART_HMI_BUTTON )
      wire#w2
      Coil( "DB368_M_UNIT_03".M_CODES_UNIT_03.Ack_M50 )
   END_RUNG
   RUNG wire#w1
      Contact( "DB2031_CYCLES_GENERAL".DRY_CYCLE.CYCLE_SELECTED )
      I_Contact( "DB2031_CYCLES_GENERAL".MANUAL_LOAD_CYCLE.CYCLE_SELECTED )
   END_RUNG wire#w2
   // the same network as SCL:
   "DB368_M_UNIT_03".M_CODES_UNIT_03.Ack_M50 := "DB368_M_UNIT_03".M_CODES_UNIT_03.M50 AND "DB8000_PART_STATUS".UNIT_03.FIXTURE_1.PART_A.STATUS.PRESENT AND "DB8000_PART_STATUS".UNIT_01.STATION_1.PART_A.STATUS.CELL_STATUS.COOLING_DONE AND ("DB8100_MANUAL_LOADING_PART_STATUS".UNIT_03_ADD_PART_HMI_BUTTON OR ("DB2031_CYCLES_GENERAL".DRY_CYCLE.CYCLE_SELECTED AND NOT "DB2031_CYCLES_GENERAL".MANUAL_LOAD_CYCLE.CYCLE_SELECTED));
END_REGION

REGION Network 40: M50-LOAD PART FROM ROBOT (READ IN DISABLE)
   RUNG wire#powerrail
      Contact( "LBP_Chan1".MDyn[50] )
      wire#w1
      I_Contact( "DB368_M_UNIT_03".M_CODES_UNIT_03.Ack_M50 )
      I_Contact( "DB2120_MPP_ITC_IPC".RESET_FAULTS )
      I_Contact( "DB368_M_UNIT_03".M_CODES_UNIT_03.M_RESET_PULSE )
      Coil( "DB368_M_UNIT_03".M_CODES_UNIT_03.M50 )
   END_RUNG
   RUNG wire#powerrail
      Contact( "DB368_M_UNIT_03".M_CODES_UNIT_03.M50 )
   END_RUNG wire#w1
   // the same network as SCL:
   "DB368_M_UNIT_03".M_CODES_UNIT_03.M50 := ("LBP_Chan1".MDyn[50] OR "DB368_M_UNIT_03".M_CODES_UNIT_03.M50) AND NOT "DB368_M_UNIT_03".M_CODES_UNIT_03.Ack_M50 AND NOT "DB2120_MPP_ITC_IPC".RESET_FAULTS AND NOT "DB368_M_UNIT_03".M_CODES_UNIT_03.M_RESET_PULSE;
END_REGION

REGION Network 41: ACKNOWLEDGE M51-UNLOAD PART FROM ROBOT (READ IN DISABLE)
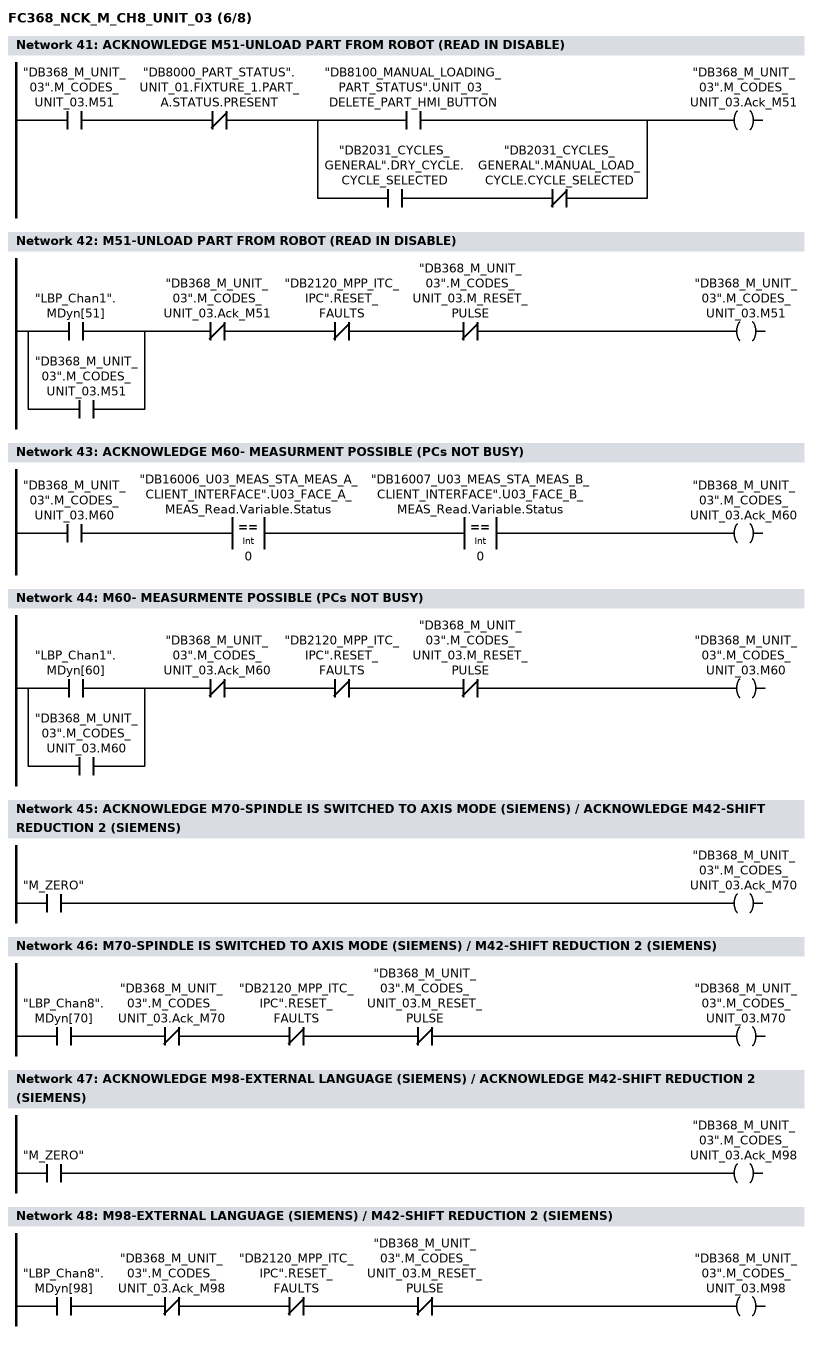
   RUNG wire#powerrail
      Contact( "DB368_M_UNIT_03".M_CODES_UNIT_03.M51 )
      I_Contact( "DB8000_PART_STATUS".UNIT_01.FIXTURE_1.PART_A.STATUS.PRESENT )
      wire#w1
      Contact( "DB8100_MANUAL_LOADING_PART_STATUS".UNIT_03_DELETE_PART_HMI_BUTTON )
      wire#w2
      Coil( "DB368_M_UNIT_03".M_CODES_UNIT_03.Ack_M51 )
   END_RUNG
   RUNG wire#w1
      Contact( "DB2031_CYCLES_GENERAL".DRY_CYCLE.CYCLE_SELECTED )
      I_Contact( "DB2031_CYCLES_GENERAL".MANUAL_LOAD_CYCLE.CYCLE_SELECTED )
   END_RUNG wire#w2
   // the same network as SCL:
   "DB368_M_UNIT_03".M_CODES_UNIT_03.Ack_M51 := "DB368_M_UNIT_03".M_CODES_UNIT_03.M51 AND NOT "DB8000_PART_STATUS".UNIT_01.FIXTURE_1.PART_A.STATUS.PRESENT AND ("DB8100_MANUAL_LOADING_PART_STATUS".UNIT_03_DELETE_PART_HMI_BUTTON OR ("DB2031_CYCLES_GENERAL".DRY_CYCLE.CYCLE_SELECTED AND NOT "DB2031_CYCLES_GENERAL".MANUAL_LOAD_CYCLE.CYCLE_SELECTED));
END_REGION

REGION Network 42: M51-UNLOAD PART FROM ROBOT (READ IN DISABLE)
   RUNG wire#powerrail
      Contact( "LBP_Chan1".MDyn[51] )
      wire#w1
      I_Contact( "DB368_M_UNIT_03".M_CODES_UNIT_03.Ack_M51 )
      I_Contact( "DB2120_MPP_ITC_IPC".RESET_FAULTS )
      I_Contact( "DB368_M_UNIT_03".M_CODES_UNIT_03.M_RESET_PULSE )
      Coil( "DB368_M_UNIT_03".M_CODES_UNIT_03.M51 )
   END_RUNG
   RUNG wire#powerrail
      Contact( "DB368_M_UNIT_03".M_CODES_UNIT_03.M51 )
   END_RUNG wire#w1
   // the same network as SCL:
   "DB368_M_UNIT_03".M_CODES_UNIT_03.M51 := ("LBP_Chan1".MDyn[51] OR "DB368_M_UNIT_03".M_CODES_UNIT_03.M51) AND NOT "DB368_M_UNIT_03".M_CODES_UNIT_03.Ack_M51 AND NOT "DB2120_MPP_ITC_IPC".RESET_FAULTS AND NOT "DB368_M_UNIT_03".M_CODES_UNIT_03.M_RESET_PULSE;
END_REGION

REGION Network 43: ACKNOWLEDGE M60- MEASURMENT POSSIBLE (PCs NOT BUSY)
   RUNG wire#powerrail
      Contact( "DB368_M_UNIT_03".M_CODES_UNIT_03.M60 )
      { S7_Templates := "SrcType := Int" } EQ_Contact(in1 := "DB16006_U03_MEAS_STA_MEAS_A_CLIENT_INTERFACE".U03_FACE_A_MEAS_Read.Variable.Status, in2 := 0)
      { S7_Templates := "SrcType := Int" } EQ_Contact(in1 := "DB16007_U03_MEAS_STA_MEAS_B_CLIENT_INTERFACE".U03_FACE_B_MEAS_Read.Variable.Status, in2 := 0)
      Coil( "DB368_M_UNIT_03".M_CODES_UNIT_03.Ack_M60 )
   END_RUNG
   // the same network as SCL:
   "DB368_M_UNIT_03".M_CODES_UNIT_03.Ack_M60 := "DB368_M_UNIT_03".M_CODES_UNIT_03.M60 AND ("DB16006_U03_MEAS_STA_MEAS_A_CLIENT_INTERFACE".U03_FACE_A_MEAS_Read.Variable.Status = 0) AND ("DB16007_U03_MEAS_STA_MEAS_B_CLIENT_INTERFACE".U03_FACE_B_MEAS_Read.Variable.Status = 0);
END_REGION

REGION Network 44: M60- MEASURMENTE POSSIBLE (PCs NOT BUSY)
   RUNG wire#powerrail
      Contact( "LBP_Chan1".MDyn[60] )
      wire#w1
      I_Contact( "DB368_M_UNIT_03".M_CODES_UNIT_03.Ack_M60 )
      I_Contact( "DB2120_MPP_ITC_IPC".RESET_FAULTS )
      I_Contact( "DB368_M_UNIT_03".M_CODES_UNIT_03.M_RESET_PULSE )
      Coil( "DB368_M_UNIT_03".M_CODES_UNIT_03.M60 )
   END_RUNG
   RUNG wire#powerrail
      Contact( "DB368_M_UNIT_03".M_CODES_UNIT_03.M60 )
   END_RUNG wire#w1
   // the same network as SCL:
   "DB368_M_UNIT_03".M_CODES_UNIT_03.M60 := ("LBP_Chan1".MDyn[60] OR "DB368_M_UNIT_03".M_CODES_UNIT_03.M60) AND NOT "DB368_M_UNIT_03".M_CODES_UNIT_03.Ack_M60 AND NOT "DB2120_MPP_ITC_IPC".RESET_FAULTS AND NOT "DB368_M_UNIT_03".M_CODES_UNIT_03.M_RESET_PULSE;
END_REGION

REGION Network 45: ACKNOWLEDGE M70-SPINDLE IS SWITCHED TO AXIS MODE (SIEMENS) / ACKNOWLEDGE M42-SHIFT REDUCTION 2 (SIEMENS)
   RUNG wire#powerrail
      Contact( "M_ZERO" )
      Coil( "DB368_M_UNIT_03".M_CODES_UNIT_03.Ack_M70 )
   END_RUNG
   // the same network as SCL:
   "DB368_M_UNIT_03".M_CODES_UNIT_03.Ack_M70 := "M_ZERO";
END_REGION

REGION Network 46: M70-SPINDLE IS SWITCHED TO AXIS MODE (SIEMENS) / M42-SHIFT REDUCTION 2 (SIEMENS)
   RUNG wire#powerrail
      Contact( "LBP_Chan8".MDyn[70] )
      I_Contact( "DB368_M_UNIT_03".M_CODES_UNIT_03.Ack_M70 )
      I_Contact( "DB2120_MPP_ITC_IPC".RESET_FAULTS )
      I_Contact( "DB368_M_UNIT_03".M_CODES_UNIT_03.M_RESET_PULSE )
      Coil( "DB368_M_UNIT_03".M_CODES_UNIT_03.M70 )
   END_RUNG
   // the same network as SCL:
   "DB368_M_UNIT_03".M_CODES_UNIT_03.M70 := "LBP_Chan8".MDyn[70] AND NOT "DB368_M_UNIT_03".M_CODES_UNIT_03.Ack_M70 AND NOT "DB2120_MPP_ITC_IPC".RESET_FAULTS AND NOT "DB368_M_UNIT_03".M_CODES_UNIT_03.M_RESET_PULSE;
END_REGION

REGION Network 47: ACKNOWLEDGE M98-EXTERNAL LANGUAGE (SIEMENS) / ACKNOWLEDGE M42-SHIFT REDUCTION 2 (SIEMENS)
   RUNG wire#powerrail
      Contact( "M_ZERO" )
      Coil( "DB368_M_UNIT_03".M_CODES_UNIT_03.Ack_M98 )
   END_RUNG
   // the same network as SCL:
   "DB368_M_UNIT_03".M_CODES_UNIT_03.Ack_M98 := "M_ZERO";
END_REGION

REGION Network 48: M98-EXTERNAL LANGUAGE (SIEMENS) / M42-SHIFT REDUCTION 2 (SIEMENS)
   RUNG wire#powerrail
      Contact( "LBP_Chan8".MDyn[98] )
      I_Contact( "DB368_M_UNIT_03".M_CODES_UNIT_03.Ack_M98 )
      I_Contact( "DB2120_MPP_ITC_IPC".RESET_FAULTS )
      I_Contact( "DB368_M_UNIT_03".M_CODES_UNIT_03.M_RESET_PULSE )
      Coil( "DB368_M_UNIT_03".M_CODES_UNIT_03.M98 )
   END_RUNG
   // the same network as SCL:
   "DB368_M_UNIT_03".M_CODES_UNIT_03.M98 := "LBP_Chan8".MDyn[98] AND NOT "DB368_M_UNIT_03".M_CODES_UNIT_03.Ack_M98 AND NOT "DB2120_MPP_ITC_IPC".RESET_FAULTS AND NOT "DB368_M_UNIT_03".M_CODES_UNIT_03.M_RESET_PULSE;
END_REGION

REGION Network 49: ACKNOWLEDGE M99-EXTERNAL LANGUAGE (SIEMENS) / ACKNOWLEDGE M42-SHIFT REDUCTION 2 (SIEMENS)
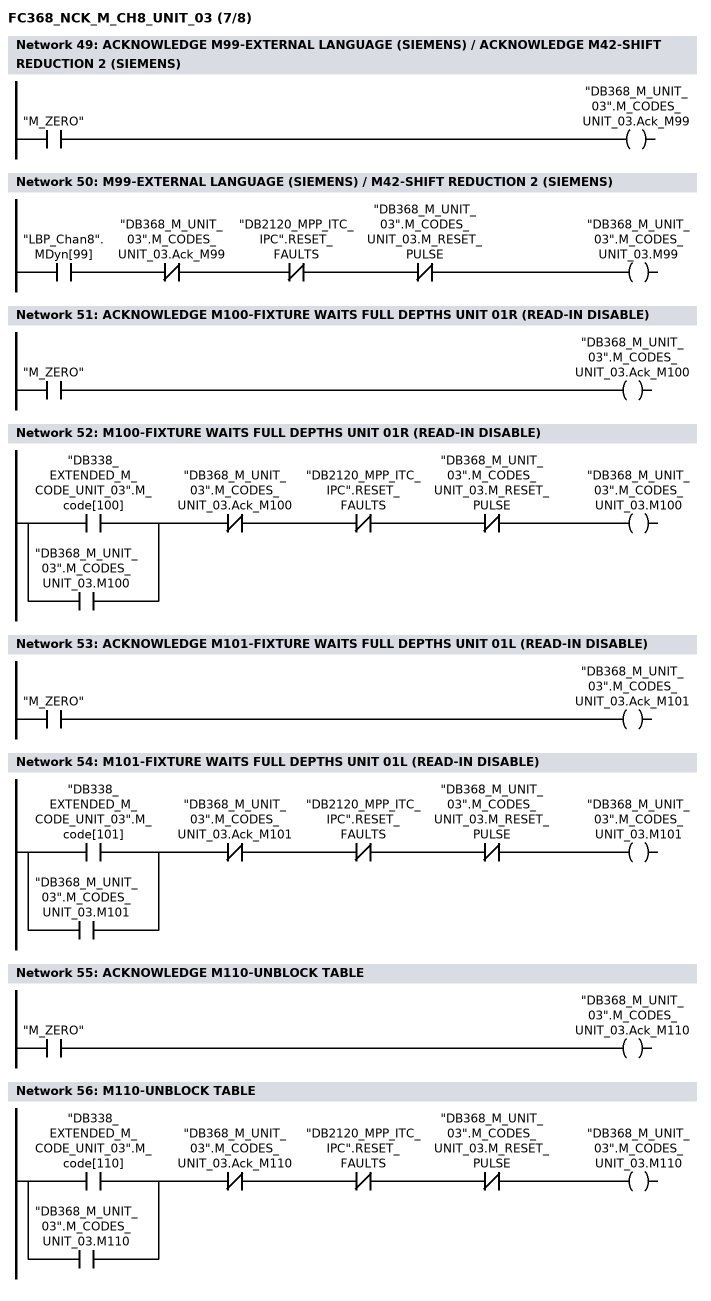
   RUNG wire#powerrail
      Contact( "M_ZERO" )
      Coil( "DB368_M_UNIT_03".M_CODES_UNIT_03.Ack_M99 )
   END_RUNG
   // the same network as SCL:
   "DB368_M_UNIT_03".M_CODES_UNIT_03.Ack_M99 := "M_ZERO";
END_REGION

REGION Network 50: M99-EXTERNAL LANGUAGE (SIEMENS) / M42-SHIFT REDUCTION 2 (SIEMENS)
   RUNG wire#powerrail
      Contact( "LBP_Chan8".MDyn[99] )
      I_Contact( "DB368_M_UNIT_03".M_CODES_UNIT_03.Ack_M99 )
      I_Contact( "DB2120_MPP_ITC_IPC".RESET_FAULTS )
      I_Contact( "DB368_M_UNIT_03".M_CODES_UNIT_03.M_RESET_PULSE )
      Coil( "DB368_M_UNIT_03".M_CODES_UNIT_03.M99 )
   END_RUNG
   // the same network as SCL:
   "DB368_M_UNIT_03".M_CODES_UNIT_03.M99 := "LBP_Chan8".MDyn[99] AND NOT "DB368_M_UNIT_03".M_CODES_UNIT_03.Ack_M99 AND NOT "DB2120_MPP_ITC_IPC".RESET_FAULTS AND NOT "DB368_M_UNIT_03".M_CODES_UNIT_03.M_RESET_PULSE;
END_REGION

REGION Network 51: ACKNOWLEDGE M100-FIXTURE WAITS FULL DEPTHS UNIT 01R (READ-IN DISABLE)
   RUNG wire#powerrail
      Contact( "M_ZERO" )
      Coil( "DB368_M_UNIT_03".M_CODES_UNIT_03.Ack_M100 )
   END_RUNG
   // the same network as SCL:
   "DB368_M_UNIT_03".M_CODES_UNIT_03.Ack_M100 := "M_ZERO";
END_REGION

REGION Network 52: M100-FIXTURE WAITS FULL DEPTHS UNIT 01R (READ-IN DISABLE)
   RUNG wire#powerrail
      Contact( "DB338_EXTENDED_M_CODE_UNIT_03".M_code[100] )
      wire#w1
      I_Contact( "DB368_M_UNIT_03".M_CODES_UNIT_03.Ack_M100 )
      I_Contact( "DB2120_MPP_ITC_IPC".RESET_FAULTS )
      I_Contact( "DB368_M_UNIT_03".M_CODES_UNIT_03.M_RESET_PULSE )
      Coil( "DB368_M_UNIT_03".M_CODES_UNIT_03.M100 )
   END_RUNG
   RUNG wire#powerrail
      Contact( "DB368_M_UNIT_03".M_CODES_UNIT_03.M100 )
   END_RUNG wire#w1
   // the same network as SCL:
   "DB368_M_UNIT_03".M_CODES_UNIT_03.M100 := ("DB338_EXTENDED_M_CODE_UNIT_03".M_code[100] OR "DB368_M_UNIT_03".M_CODES_UNIT_03.M100) AND NOT "DB368_M_UNIT_03".M_CODES_UNIT_03.Ack_M100 AND NOT "DB2120_MPP_ITC_IPC".RESET_FAULTS AND NOT "DB368_M_UNIT_03".M_CODES_UNIT_03.M_RESET_PULSE;
END_REGION

REGION Network 53: ACKNOWLEDGE M101-FIXTURE WAITS FULL DEPTHS UNIT 01L (READ-IN DISABLE)
   RUNG wire#powerrail
      Contact( "M_ZERO" )
      Coil( "DB368_M_UNIT_03".M_CODES_UNIT_03.Ack_M101 )
   END_RUNG
   // the same network as SCL:
   "DB368_M_UNIT_03".M_CODES_UNIT_03.Ack_M101 := "M_ZERO";
END_REGION

REGION Network 54: M101-FIXTURE WAITS FULL DEPTHS UNIT 01L (READ-IN DISABLE)
   RUNG wire#powerrail
      Contact( "DB338_EXTENDED_M_CODE_UNIT_03".M_code[101] )
      wire#w1
      I_Contact( "DB368_M_UNIT_03".M_CODES_UNIT_03.Ack_M101 )
      I_Contact( "DB2120_MPP_ITC_IPC".RESET_FAULTS )
      I_Contact( "DB368_M_UNIT_03".M_CODES_UNIT_03.M_RESET_PULSE )
      Coil( "DB368_M_UNIT_03".M_CODES_UNIT_03.M101 )
   END_RUNG
   RUNG wire#powerrail
      Contact( "DB368_M_UNIT_03".M_CODES_UNIT_03.M101 )
   END_RUNG wire#w1
   // the same network as SCL:
   "DB368_M_UNIT_03".M_CODES_UNIT_03.M101 := ("DB338_EXTENDED_M_CODE_UNIT_03".M_code[101] OR "DB368_M_UNIT_03".M_CODES_UNIT_03.M101) AND NOT "DB368_M_UNIT_03".M_CODES_UNIT_03.Ack_M101 AND NOT "DB2120_MPP_ITC_IPC".RESET_FAULTS AND NOT "DB368_M_UNIT_03".M_CODES_UNIT_03.M_RESET_PULSE;
END_REGION

REGION Network 55: ACKNOWLEDGE M110-UNBLOCK TABLE
   RUNG wire#powerrail
      Contact( "M_ZERO" )
      Coil( "DB368_M_UNIT_03".M_CODES_UNIT_03.Ack_M110 )
   END_RUNG
   // the same network as SCL:
   "DB368_M_UNIT_03".M_CODES_UNIT_03.Ack_M110 := "M_ZERO";
END_REGION

REGION Network 56: M110-UNBLOCK TABLE
   RUNG wire#powerrail
      Contact( "DB338_EXTENDED_M_CODE_UNIT_03".M_code[110] )
      wire#w1
      I_Contact( "DB368_M_UNIT_03".M_CODES_UNIT_03.Ack_M110 )
      I_Contact( "DB2120_MPP_ITC_IPC".RESET_FAULTS )
      I_Contact( "DB368_M_UNIT_03".M_CODES_UNIT_03.M_RESET_PULSE )
      Coil( "DB368_M_UNIT_03".M_CODES_UNIT_03.M110 )
   END_RUNG
   RUNG wire#powerrail
      Contact( "DB368_M_UNIT_03".M_CODES_UNIT_03.M110 )
   END_RUNG wire#w1
   // the same network as SCL:
   "DB368_M_UNIT_03".M_CODES_UNIT_03.M110 := ("DB338_EXTENDED_M_CODE_UNIT_03".M_code[110] OR "DB368_M_UNIT_03".M_CODES_UNIT_03.M110) AND NOT "DB368_M_UNIT_03".M_CODES_UNIT_03.Ack_M110 AND NOT "DB2120_MPP_ITC_IPC".RESET_FAULTS AND NOT "DB368_M_UNIT_03".M_CODES_UNIT_03.M_RESET_PULSE;
END_REGION

REGION Network 57: ACKNOWLEDGE M111-BLOCK TABLE
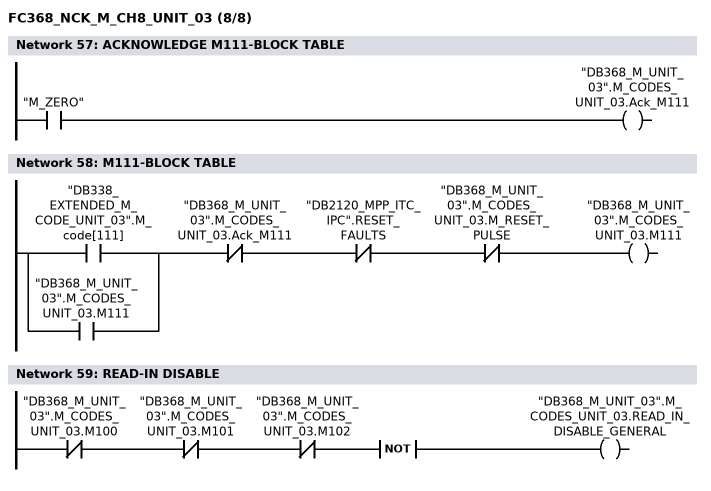
   RUNG wire#powerrail
      Contact( "M_ZERO" )
      Coil( "DB368_M_UNIT_03".M_CODES_UNIT_03.Ack_M111 )
   END_RUNG
   // the same network as SCL:
   "DB368_M_UNIT_03".M_CODES_UNIT_03.Ack_M111 := "M_ZERO";
END_REGION

REGION Network 58: M111-BLOCK TABLE
   RUNG wire#powerrail
      Contact( "DB338_EXTENDED_M_CODE_UNIT_03".M_code[111] )
      wire#w1
      I_Contact( "DB368_M_UNIT_03".M_CODES_UNIT_03.Ack_M111 )
      I_Contact( "DB2120_MPP_ITC_IPC".RESET_FAULTS )
      I_Contact( "DB368_M_UNIT_03".M_CODES_UNIT_03.M_RESET_PULSE )
      Coil( "DB368_M_UNIT_03".M_CODES_UNIT_03.M111 )
   END_RUNG
   RUNG wire#powerrail
      Contact( "DB368_M_UNIT_03".M_CODES_UNIT_03.M111 )
   END_RUNG wire#w1
   // the same network as SCL:
   "DB368_M_UNIT_03".M_CODES_UNIT_03.M111 := ("DB338_EXTENDED_M_CODE_UNIT_03".M_code[111] OR "DB368_M_UNIT_03".M_CODES_UNIT_03.M111) AND NOT "DB368_M_UNIT_03".M_CODES_UNIT_03.Ack_M111 AND NOT "DB2120_MPP_ITC_IPC".RESET_FAULTS AND NOT "DB368_M_UNIT_03".M_CODES_UNIT_03.M_RESET_PULSE;
END_REGION

REGION Network 59: READ-IN DISABLE
   RUNG wire#powerrail
      I_Contact( "DB368_M_UNIT_03".M_CODES_UNIT_03.M100 )
      I_Contact( "DB368_M_UNIT_03".M_CODES_UNIT_03.M101 )
      I_Contact( "DB368_M_UNIT_03".M_CODES_UNIT_03.M102 )
      Not()
      Coil( "DB368_M_UNIT_03".M_CODES_UNIT_03.READ_IN_DISABLE_GENERAL )
   END_RUNG
   // the same network as SCL:
   "DB368_M_UNIT_03".M_CODES_UNIT_03.READ_IN_DISABLE_GENERAL := NOT (NOT "DB368_M_UNIT_03".M_CODES_UNIT_03.M100 AND NOT "DB368_M_UNIT_03".M_CODES_UNIT_03.M101 AND NOT "DB368_M_UNIT_03".M_CODES_UNIT_03.M102);
END_REGION
END_FUNCTION
